TYPE "UDT_WSVStatistics"
VERSION : 0.1
   STRUCT
      "010" { ExternalAccessible := 'False'; ExternalVisible := 'False'; ExternalWritable := 'False'} : Struct
         Conveyor { ExternalAccessible := 'False'; ExternalVisible := 'False'; ExternalWritable := 'False'; S7_SetPoint := 'False'} : "UDT_ConveyorStatistics";
         MCO_M01 { ExternalAccessible := 'False'; ExternalVisible := 'False'; ExternalWritable := 'False'; S7_SetPoint := 'False'} : "UDT_VfdStatistics";
      END_STRUCT;
      "020" { ExternalAccessible := 'False'; ExternalVisible := 'False'; ExternalWritable := 'False'} : Struct
         Conveyor { ExternalAccessible := 'False'; ExternalVisible := 'False'; ExternalWritable := 'False'; S7_SetPoint := 'False'} : "UDT_ConveyorStatistics";
         PEC_Eos { ExternalAccessible := 'False'; ExternalVisible := 'False'; ExternalWritable := 'False'} : "UDT_PECStatistics";
         MCO_M01 { ExternalAccessible := 'False'; ExternalVisible := 'False'; ExternalWritable := 'False'; S7_SetPoint := 'False'} : "UDT_VfdStatistics";
      END_STRUCT;
      "030" { ExternalAccessible := 'False'; ExternalVisible := 'False'; ExternalWritable := 'False'} : Struct
         Conveyor { ExternalAccessible := 'False'; ExternalVisible := 'False'; ExternalWritable := 'False'; S7_SetPoint := 'False'} : "UDT_ConveyorStatistics";
         PEC_Eos { ExternalAccessible := 'False'; ExternalVisible := 'False'; ExternalWritable := 'False'} : "UDT_PECStatistics";
         MCO_M01 { ExternalAccessible := 'False'; ExternalVisible := 'False'; ExternalWritable := 'False'; S7_SetPoint := 'False'} : "UDT_VfdStatistics";
      END_STRUCT;
      "040" { ExternalAccessible := 'False'; ExternalVisible := 'False'; ExternalWritable := 'False'} : Struct
         Conveyor { ExternalAccessible := 'False'; ExternalVisible := 'False'; ExternalWritable := 'False'; S7_SetPoint := 'False'} : "UDT_ConveyorStatistics";
         PEC_Eos { ExternalAccessible := 'False'; ExternalVisible := 'False'; ExternalWritable := 'False'} : "UDT_PECStatistics";
         MCO_M01 { ExternalAccessible := 'False'; ExternalVisible := 'False'; ExternalWritable := 'False'; S7_SetPoint := 'False'} : "UDT_VfdStatistics";
      END_STRUCT;
      "050" { ExternalAccessible := 'False'; ExternalVisible := 'False'; ExternalWritable := 'False'} : Struct
         Conveyor { ExternalAccessible := 'False'; ExternalVisible := 'False'; ExternalWritable := 'False'; S7_SetPoint := 'False'} : "UDT_ConveyorStatistics";
         PEC_Eos { ExternalAccessible := 'False'; ExternalVisible := 'False'; ExternalWritable := 'False'} : "UDT_PECStatistics";
         MCO_M01 { ExternalAccessible := 'False'; ExternalVisible := 'False'; ExternalWritable := 'False'; S7_SetPoint := 'False'} : "UDT_VfdStatistics";
      END_STRUCT;
      "060" { ExternalAccessible := 'False'; ExternalVisible := 'False'; ExternalWritable := 'False'} : Struct
         Conveyor { ExternalAccessible := 'False'; ExternalVisible := 'False'; ExternalWritable := 'False'; S7_SetPoint := 'False'} : "UDT_ConveyorStatistics";
         PEC_Eos { ExternalAccessible := 'False'; ExternalVisible := 'False'; ExternalWritable := 'False'} : "UDT_PECStatistics";
         MCO_M01 { ExternalAccessible := 'False'; ExternalVisible := 'False'; ExternalWritable := 'False'; S7_SetPoint := 'False'} : "UDT_VfdStatistics";
      END_STRUCT;
      "070" { ExternalAccessible := 'False'; ExternalVisible := 'False'; ExternalWritable := 'False'} : Struct
         Conveyor { ExternalAccessible := 'False'; ExternalVisible := 'False'; ExternalWritable := 'False'; S7_SetPoint := 'False'} : "UDT_ConveyorStatistics";
         PEC_Eos { ExternalAccessible := 'False'; ExternalVisible := 'False'; ExternalWritable := 'False'} : "UDT_PECStatistics";
         MCO_M01 { ExternalAccessible := 'False'; ExternalVisible := 'False'; ExternalWritable := 'False'; S7_SetPoint := 'False'} : "UDT_VfdStatistics";
      END_STRUCT;
      "080" { ExternalAccessible := 'False'; ExternalVisible := 'False'; ExternalWritable := 'False'} : Struct
         Conveyor { ExternalAccessible := 'False'; ExternalVisible := 'False'; ExternalWritable := 'False'; S7_SetPoint := 'False'} : "UDT_ConveyorStatistics";
         PEC_Eos { ExternalAccessible := 'False'; ExternalVisible := 'False'; ExternalWritable := 'False'} : "UDT_PECStatistics";
         MCO_M01 { ExternalAccessible := 'False'; ExternalVisible := 'False'; ExternalWritable := 'False'; S7_SetPoint := 'False'} : "UDT_VfdStatistics";
      END_STRUCT;
      "090" { ExternalAccessible := 'False'; ExternalVisible := 'False'; ExternalWritable := 'False'} : Struct
         Conveyor { ExternalAccessible := 'False'; ExternalVisible := 'False'; ExternalWritable := 'False'; S7_SetPoint := 'False'} : "UDT_ConveyorStatistics";
         MCO_M01 { ExternalAccessible := 'False'; ExternalVisible := 'False'; ExternalWritable := 'False'; S7_SetPoint := 'False'} : "UDT_VfdStatistics";
      END_STRUCT;
      "100" { ExternalAccessible := 'False'; ExternalVisible := 'False'; ExternalWritable := 'False'} : Struct
         Conveyor { ExternalAccessible := 'False'; ExternalVisible := 'False'; ExternalWritable := 'False'; S7_SetPoint := 'False'} : "UDT_ConveyorStatistics";
         PEC_Eos { ExternalAccessible := 'False'; ExternalVisible := 'False'; ExternalWritable := 'False'} : "UDT_PECStatistics";
         MCO_M01 { ExternalAccessible := 'False'; ExternalVisible := 'False'; ExternalWritable := 'False'; S7_SetPoint := 'False'} : "UDT_VfdStatistics";
      END_STRUCT;
      "110" { ExternalAccessible := 'False'; ExternalVisible := 'False'; ExternalWritable := 'False'} : Struct
         Conveyor { ExternalAccessible := 'False'; ExternalVisible := 'False'; ExternalWritable := 'False'; S7_SetPoint := 'False'} : "UDT_ConveyorStatistics";
         PEC_Eos { ExternalAccessible := 'False'; ExternalVisible := 'False'; ExternalWritable := 'False'} : "UDT_PECStatistics";
         MCO_M01 { ExternalAccessible := 'False'; ExternalVisible := 'False'; ExternalWritable := 'False'; S7_SetPoint := 'False'} : "UDT_VfdStatistics";
      END_STRUCT;
      "120" { ExternalAccessible := 'False'; ExternalVisible := 'False'; ExternalWritable := 'False'} : Struct
         Conveyor { ExternalAccessible := 'False'; ExternalVisible := 'False'; ExternalWritable := 'False'; S7_SetPoint := 'False'} : "UDT_ConveyorStatistics";
         PEC_Eos { ExternalAccessible := 'False'; ExternalVisible := 'False'; ExternalWritable := 'False'} : "UDT_PECStatistics";
         MCO_M01 { ExternalAccessible := 'False'; ExternalVisible := 'False'; ExternalWritable := 'False'; S7_SetPoint := 'False'} : "UDT_VfdStatistics";
      END_STRUCT;
      "121" { ExternalAccessible := 'False'; ExternalVisible := 'False'; ExternalWritable := 'False'} : Struct
         RightAngledTransfer { ExternalAccessible := 'False'; ExternalVisible := 'False'; ExternalWritable := 'False'; S7_SetPoint := 'False'} : "UDT_RATStatistics";
         MCO_M01 { ExternalAccessible := 'False'; ExternalVisible := 'False'; ExternalWritable := 'False'} : "UDT_VfdStatistics";
      END_STRUCT;
      "230" { ExternalAccessible := 'False'; ExternalVisible := 'False'; ExternalWritable := 'False'} : Struct
         Conveyor { ExternalAccessible := 'False'; ExternalVisible := 'False'; ExternalWritable := 'False'; S7_SetPoint := 'False'} : "UDT_ConveyorStatistics";
         PEC_Eos { ExternalAccessible := 'False'; ExternalVisible := 'False'; ExternalWritable := 'False'} : "UDT_PECUpdateStatistics";
         MCO_M01 { ExternalAccessible := 'False'; ExternalVisible := 'False'; ExternalWritable := 'False'; S7_SetPoint := 'False'} : "UDT_VfdStatistics";
      END_STRUCT;
      "240" { ExternalAccessible := 'False'; ExternalVisible := 'False'; ExternalWritable := 'False'} : Struct
         Conveyor { ExternalAccessible := 'False'; ExternalVisible := 'False'; ExternalWritable := 'False'; S7_SetPoint := 'False'} : "UDT_ConveyorStatistics";
         PEC_Eos { ExternalAccessible := 'False'; ExternalVisible := 'False'; ExternalWritable := 'False'; S7_SetPoint := 'False'} : "UDT_PECStatistics";
         MCO_M01 { ExternalAccessible := 'False'; ExternalVisible := 'False'; ExternalWritable := 'False'; S7_SetPoint := 'False'} : "UDT_VfdStatistics";
      END_STRUCT;
      "241" { ExternalAccessible := 'False'; ExternalVisible := 'False'; ExternalWritable := 'False'} : Struct
         RightAngledTransfer { ExternalAccessible := 'False'; ExternalVisible := 'False'; ExternalWritable := 'False'} : "UDT_RATStatistics";
         MCO_M01 { ExternalAccessible := 'False'; ExternalVisible := 'False'; ExternalWritable := 'False'} : "UDT_VfdStatistics";
      END_STRUCT;
      "250" { ExternalAccessible := 'False'; ExternalVisible := 'False'; ExternalWritable := 'False'} : Struct
         Conveyor { ExternalAccessible := 'False'; ExternalVisible := 'False'; ExternalWritable := 'False'} : "UDT_ConveyorStatistics";
         PEC_EoS { ExternalAccessible := 'False'; ExternalVisible := 'False'; ExternalWritable := 'False'; S7_SetPoint := 'False'} : "UDT_PECUpdateStatistics";
         MCO_M01 { ExternalAccessible := 'False'; ExternalVisible := 'False'; ExternalWritable := 'False'; S7_SetPoint := 'False'} : "UDT_VfdStatistics";
      END_STRUCT;
      "260" { ExternalAccessible := 'False'; ExternalVisible := 'False'; ExternalWritable := 'False'} : Struct
         Conveyor { ExternalAccessible := 'False'; ExternalVisible := 'False'; ExternalWritable := 'False'} : "UDT_ConveyorStatistics";
         VFD { ExternalAccessible := 'False'; ExternalVisible := 'False'; ExternalWritable := 'False'; S7_SetPoint := 'False'} : "UDT_VfdStatistics";
      END_STRUCT;
      "270" { ExternalAccessible := 'False'; ExternalVisible := 'False'; ExternalWritable := 'False'} : Struct
         Conveyor { ExternalAccessible := 'False'; ExternalVisible := 'False'; ExternalWritable := 'False'} : "UDT_ConveyorStatistics";
         PEC_EoS { ExternalAccessible := 'False'; ExternalVisible := 'False'; ExternalWritable := 'False'; S7_SetPoint := 'False'} : "UDT_PECStatistics";
         MCO_M01 { ExternalAccessible := 'False'; ExternalVisible := 'False'; ExternalWritable := 'False'; S7_SetPoint := 'False'} : "UDT_VfdStatistics";
      END_STRUCT;
      "280" { ExternalAccessible := 'False'; ExternalVisible := 'False'; ExternalWritable := 'False'} : Struct
         Conveyor { ExternalAccessible := 'False'; ExternalVisible := 'False'; ExternalWritable := 'False'} : "UDT_ConveyorStatistics";
         PEC_EoS { ExternalAccessible := 'False'; ExternalVisible := 'False'; ExternalWritable := 'False'; S7_SetPoint := 'False'} : "UDT_PECStatistics";
         MCO_M01 { ExternalAccessible := 'False'; ExternalVisible := 'False'; ExternalWritable := 'False'} : "UDT_VfdStatistics";
      END_STRUCT;
      "310" { ExternalAccessible := 'False'; ExternalVisible := 'False'; ExternalWritable := 'False'} : Struct
         Conveyor { ExternalAccessible := 'False'; ExternalVisible := 'False'; ExternalWritable := 'False'; S7_SetPoint := 'False'} : "UDT_ConveyorStatistics";
         VFD { ExternalAccessible := 'False'; ExternalVisible := 'False'; ExternalWritable := 'False'; S7_SetPoint := 'False'} : "UDT_VfdStatistics";
      END_STRUCT;
      "320" { ExternalAccessible := 'False'; ExternalVisible := 'False'; ExternalWritable := 'False'} : Struct
         Conveyor { ExternalAccessible := 'False'; ExternalVisible := 'False'; ExternalWritable := 'False'; S7_SetPoint := 'False'} : "UDT_ConveyorStatistics";
         PEC_Eos { ExternalAccessible := 'False'; ExternalVisible := 'False'; ExternalWritable := 'False'} : "UDT_PECUpdateStatistics";
         MCO_M01 { ExternalAccessible := 'False'; ExternalVisible := 'False'; ExternalWritable := 'False'; S7_SetPoint := 'False'} : "UDT_VfdStatistics";
      END_STRUCT;
      "330" { ExternalAccessible := 'False'; ExternalVisible := 'False'; ExternalWritable := 'False'} : Struct
         Conveyor { ExternalAccessible := 'False'; ExternalVisible := 'False'; ExternalWritable := 'False'; S7_SetPoint := 'False'} : "UDT_ConveyorStatistics";
         PEC_Eos { ExternalAccessible := 'False'; ExternalVisible := 'False'; ExternalWritable := 'False'} : "UDT_PECUpdateStatistics";
         MCO_M01 { ExternalAccessible := 'False'; ExternalVisible := 'False'; ExternalWritable := 'False'} : "UDT_VfdStatistics";
      END_STRUCT;
      "340" { ExternalAccessible := 'False'; ExternalVisible := 'False'; ExternalWritable := 'False'} : Struct
         Conveyor { ExternalAccessible := 'False'; ExternalVisible := 'False'; ExternalWritable := 'False'; S7_SetPoint := 'False'} : "UDT_ConveyorStatistics";
         PEC_Eos { ExternalAccessible := 'False'; ExternalVisible := 'False'; ExternalWritable := 'False'} : "UDT_PECStatistics";
         MCO_M01 { ExternalAccessible := 'False'; ExternalVisible := 'False'; ExternalWritable := 'False'; S7_SetPoint := 'False'} : "UDT_VfdStatistics";
      END_STRUCT;
      "341" { ExternalAccessible := 'False'; ExternalVisible := 'False'; ExternalWritable := 'False'} : Struct
         RightAngledTransfer { ExternalAccessible := 'False'; ExternalVisible := 'False'; ExternalWritable := 'False'; S7_SetPoint := 'False'} : "UDT_RATStatistics";
         MCO_M01 { ExternalAccessible := 'False'; ExternalVisible := 'False'; ExternalWritable := 'False'} : "UDT_VfdStatistics";
      END_STRUCT;
      "350" { ExternalAccessible := 'False'; ExternalVisible := 'False'; ExternalWritable := 'False'} : Struct
         Conveyor { ExternalAccessible := 'False'; ExternalVisible := 'False'; ExternalWritable := 'False'; S7_SetPoint := 'False'} : "UDT_ConveyorStatistics";
         PEC_Eos { ExternalAccessible := 'False'; ExternalVisible := 'False'; ExternalWritable := 'False'} : "UDT_PECStatistics";
         MCO_M01 { ExternalAccessible := 'False'; ExternalVisible := 'False'; ExternalWritable := 'False'; S7_SetPoint := 'False'} : "UDT_VfdStatistics";
      END_STRUCT;
      "351" { ExternalAccessible := 'False'; ExternalVisible := 'False'; ExternalWritable := 'False'} : Struct
         RightAngledTransfer { ExternalAccessible := 'False'; ExternalVisible := 'False'; ExternalWritable := 'False'; S7_SetPoint := 'False'} : "UDT_RATStatistics";
         MCO_M01 { ExternalAccessible := 'False'; ExternalVisible := 'False'; ExternalWritable := 'False'} : "UDT_VfdStatistics";
      END_STRUCT;
      "360" { ExternalAccessible := 'False'; ExternalVisible := 'False'; ExternalWritable := 'False'} : Struct
         Conveyor { ExternalAccessible := 'False'; ExternalVisible := 'False'; ExternalWritable := 'False'; S7_SetPoint := 'False'} : "UDT_ConveyorStatistics";
         PEC_Eos { ExternalAccessible := 'False'; ExternalVisible := 'False'; ExternalWritable := 'False'} : "UDT_PECStatistics";
         MCO_M01 { ExternalAccessible := 'False'; ExternalVisible := 'False'; ExternalWritable := 'False'; S7_SetPoint := 'False'} : "UDT_VfdStatistics";
      END_STRUCT;
      "361" { ExternalAccessible := 'False'; ExternalVisible := 'False'; ExternalWritable := 'False'} : Struct
         RightAngledTransfer { ExternalAccessible := 'False'; ExternalVisible := 'False'; ExternalWritable := 'False'; S7_SetPoint := 'False'} : "UDT_RATStatistics";
         MCO_M01 { ExternalAccessible := 'False'; ExternalVisible := 'False'; ExternalWritable := 'False'} : "UDT_VfdStatistics";
      END_STRUCT;
      "370" { ExternalAccessible := 'False'; ExternalVisible := 'False'; ExternalWritable := 'False'} : Struct
         Conveyor { ExternalAccessible := 'False'; ExternalVisible := 'False'; ExternalWritable := 'False'; S7_SetPoint := 'False'} : "UDT_ConveyorStatistics";
         PEC_Eos { ExternalAccessible := 'False'; ExternalVisible := 'False'; ExternalWritable := 'False'} : "UDT_PECStatistics";
         MCO_M01 { ExternalAccessible := 'False'; ExternalVisible := 'False'; ExternalWritable := 'False'; S7_SetPoint := 'False'} : "UDT_VfdStatistics";
      END_STRUCT;
      "371" { ExternalAccessible := 'False'; ExternalVisible := 'False'; ExternalWritable := 'False'} : Struct
         RightAngledTransfer { ExternalAccessible := 'False'; ExternalVisible := 'False'; ExternalWritable := 'False'; S7_SetPoint := 'False'} : "UDT_RATStatistics";
         MCO_M01 { ExternalAccessible := 'False'; ExternalVisible := 'False'; ExternalWritable := 'False'} : "UDT_VfdStatistics";
      END_STRUCT;
      "380" { ExternalAccessible := 'False'; ExternalVisible := 'False'; ExternalWritable := 'False'} : Struct
         Conveyor { ExternalAccessible := 'False'; ExternalVisible := 'False'; ExternalWritable := 'False'; S7_SetPoint := 'False'} : "UDT_ConveyorStatistics";
         PEC_Eos { ExternalAccessible := 'False'; ExternalVisible := 'False'; ExternalWritable := 'False'} : "UDT_PECUpdateStatistics";
         MCO_M01 { ExternalAccessible := 'False'; ExternalVisible := 'False'; ExternalWritable := 'False'; S7_SetPoint := 'False'} : "UDT_VfdStatistics";
      END_STRUCT;
      "390" { ExternalAccessible := 'False'; ExternalVisible := 'False'; ExternalWritable := 'False'} : Struct
         Conveyor { ExternalAccessible := 'False'; ExternalVisible := 'False'; ExternalWritable := 'False'; S7_SetPoint := 'False'} : "UDT_ConveyorStatistics";
         PEC_Eos { ExternalAccessible := 'False'; ExternalVisible := 'False'; ExternalWritable := 'False'} : "UDT_PECUpdateStatistics";
         MCO_M01 { ExternalAccessible := 'False'; ExternalVisible := 'False'; ExternalWritable := 'False'; S7_SetPoint := 'False'} : "UDT_VfdStatistics";
      END_STRUCT;
      "530" { ExternalAccessible := 'False'; ExternalVisible := 'False'; ExternalWritable := 'False'} : Struct
         Conveyor { ExternalAccessible := 'False'; ExternalVisible := 'False'; ExternalWritable := 'False'; S7_SetPoint := 'False'} : "UDT_ConveyorStatistics";
         PEC_Eos { ExternalAccessible := 'False'; ExternalVisible := 'False'; ExternalWritable := 'False'} : "UDT_PECUpdateStatistics";
         MCO_M01 { ExternalAccessible := 'False'; ExternalVisible := 'False'; ExternalWritable := 'False'; S7_SetPoint := 'False'} : "UDT_VfdStatistics";
      END_STRUCT;
      "540" { ExternalAccessible := 'False'; ExternalVisible := 'False'; ExternalWritable := 'False'} : Struct
         Conveyor { ExternalAccessible := 'False'; ExternalVisible := 'False'; ExternalWritable := 'False'; S7_SetPoint := 'False'} : "UDT_ConveyorStatistics";
         PEC_Eos { ExternalAccessible := 'False'; ExternalVisible := 'False'; ExternalWritable := 'False'; S7_SetPoint := 'False'} : "UDT_PECStatistics";
         MCO_M01 { ExternalAccessible := 'False'; ExternalVisible := 'False'; ExternalWritable := 'False'; S7_SetPoint := 'False'} : "UDT_VfdStatistics";
      END_STRUCT;
      "541" { ExternalAccessible := 'False'; ExternalVisible := 'False'; ExternalWritable := 'False'} : Struct
         RightAngledTransfer { ExternalAccessible := 'False'; ExternalVisible := 'False'; ExternalWritable := 'False'} : "UDT_RATStatistics";
         MCO_M01 { ExternalAccessible := 'False'; ExternalVisible := 'False'; ExternalWritable := 'False'} : "UDT_VfdStatistics";
      END_STRUCT;
      "550" { ExternalAccessible := 'False'; ExternalVisible := 'False'; ExternalWritable := 'False'} : Struct
         Conveyor { ExternalAccessible := 'False'; ExternalVisible := 'False'; ExternalWritable := 'False'} : "UDT_ConveyorStatistics";
         PEC_EoS { ExternalAccessible := 'False'; ExternalVisible := 'False'; ExternalWritable := 'False'; S7_SetPoint := 'False'} : "UDT_PECUpdateStatistics";
         MCO_M01 { ExternalAccessible := 'False'; ExternalVisible := 'False'; ExternalWritable := 'False'; S7_SetPoint := 'False'} : "UDT_VfdStatistics";
      END_STRUCT;
      "560" { ExternalAccessible := 'False'; ExternalVisible := 'False'; ExternalWritable := 'False'} : Struct
         Conveyor { ExternalAccessible := 'False'; ExternalVisible := 'False'; ExternalWritable := 'False'} : "UDT_ConveyorStatistics";
         VFD { ExternalAccessible := 'False'; ExternalVisible := 'False'; ExternalWritable := 'False'; S7_SetPoint := 'False'} : "UDT_VfdStatistics";
      END_STRUCT;
      "570" { ExternalAccessible := 'False'; ExternalVisible := 'False'; ExternalWritable := 'False'} : Struct
         Conveyor { ExternalAccessible := 'False'; ExternalVisible := 'False'; ExternalWritable := 'False'} : "UDT_ConveyorStatistics";
         PEC_EoS { ExternalAccessible := 'False'; ExternalVisible := 'False'; ExternalWritable := 'False'; S7_SetPoint := 'False'} : "UDT_PECStatistics";
         MCO_M01 { ExternalAccessible := 'False'; ExternalVisible := 'False'; ExternalWritable := 'False'; S7_SetPoint := 'False'} : "UDT_VfdStatistics";
      END_STRUCT;
      "580" { ExternalAccessible := 'False'; ExternalVisible := 'False'; ExternalWritable := 'False'} : Struct
         Conveyor { ExternalAccessible := 'False'; ExternalVisible := 'False'; ExternalWritable := 'False'} : "UDT_ConveyorStatistics";
         PEC_EoS { ExternalAccessible := 'False'; ExternalVisible := 'False'; ExternalWritable := 'False'; S7_SetPoint := 'False'} : "UDT_PECStatistics";
         MCO_M01 { ExternalAccessible := 'False'; ExternalVisible := 'False'; ExternalWritable := 'False'} : "UDT_VfdStatistics";
      END_STRUCT;
      "610" { ExternalAccessible := 'False'; ExternalVisible := 'False'; ExternalWritable := 'False'} : Struct
         Conveyor { ExternalAccessible := 'False'; ExternalVisible := 'False'; ExternalWritable := 'False'; S7_SetPoint := 'False'} : "UDT_ConveyorStatistics";
         VFD { ExternalAccessible := 'False'; ExternalVisible := 'False'; ExternalWritable := 'False'; S7_SetPoint := 'False'} : "UDT_VfdStatistics";
      END_STRUCT;
      "620" { ExternalAccessible := 'False'; ExternalVisible := 'False'; ExternalWritable := 'False'} : Struct
         Conveyor { ExternalAccessible := 'False'; ExternalVisible := 'False'; ExternalWritable := 'False'; S7_SetPoint := 'False'} : "UDT_ConveyorStatistics";
         PEC_Eos { ExternalAccessible := 'False'; ExternalVisible := 'False'; ExternalWritable := 'False'} : "UDT_PECUpdateStatistics";
         MCO_M01 { ExternalAccessible := 'False'; ExternalVisible := 'False'; ExternalWritable := 'False'; S7_SetPoint := 'False'} : "UDT_VfdStatistics";
      END_STRUCT;
      "630" { ExternalAccessible := 'False'; ExternalVisible := 'False'; ExternalWritable := 'False'} : Struct
         Conveyor { ExternalAccessible := 'False'; ExternalVisible := 'False'; ExternalWritable := 'False'; S7_SetPoint := 'False'} : "UDT_ConveyorStatistics";
         PEC_Eos { ExternalAccessible := 'False'; ExternalVisible := 'False'; ExternalWritable := 'False'} : "UDT_PECUpdateStatistics";
         MCO_M01 { ExternalAccessible := 'False'; ExternalVisible := 'False'; ExternalWritable := 'False'} : "UDT_VfdStatistics";
      END_STRUCT;
      "640" { ExternalAccessible := 'False'; ExternalVisible := 'False'; ExternalWritable := 'False'} : Struct
         Conveyor { ExternalAccessible := 'False'; ExternalVisible := 'False'; ExternalWritable := 'False'; S7_SetPoint := 'False'} : "UDT_ConveyorStatistics";
         PEC_Eos { ExternalAccessible := 'False'; ExternalVisible := 'False'; ExternalWritable := 'False'} : "UDT_PECStatistics";
         MCO_M01 { ExternalAccessible := 'False'; ExternalVisible := 'False'; ExternalWritable := 'False'; S7_SetPoint := 'False'} : "UDT_VfdStatistics";
      END_STRUCT;
      "641" { ExternalAccessible := 'False'; ExternalVisible := 'False'; ExternalWritable := 'False'} : Struct
         RightAngledTransfer { ExternalAccessible := 'False'; ExternalVisible := 'False'; ExternalWritable := 'False'; S7_SetPoint := 'False'} : "UDT_RATStatistics";
         MCO_M01 { ExternalAccessible := 'False'; ExternalVisible := 'False'; ExternalWritable := 'False'} : "UDT_VfdStatistics";
      END_STRUCT;
      "650" { ExternalAccessible := 'False'; ExternalVisible := 'False'; ExternalWritable := 'False'} : Struct
         Conveyor { ExternalAccessible := 'False'; ExternalVisible := 'False'; ExternalWritable := 'False'; S7_SetPoint := 'False'} : "UDT_ConveyorStatistics";
         PEC_Eos { ExternalAccessible := 'False'; ExternalVisible := 'False'; ExternalWritable := 'False'} : "UDT_PECStatistics";
         MCO_M01 { ExternalAccessible := 'False'; ExternalVisible := 'False'; ExternalWritable := 'False'} : "UDT_VfdStatistics";
      END_STRUCT;
      "651" { ExternalAccessible := 'False'; ExternalVisible := 'False'; ExternalWritable := 'False'} : Struct
         RightAngledTransfer { ExternalAccessible := 'False'; ExternalVisible := 'False'; ExternalWritable := 'False'; S7_SetPoint := 'False'} : "UDT_RATStatistics";
         MCO_M01 { ExternalAccessible := 'False'; ExternalVisible := 'False'; ExternalWritable := 'False'} : "UDT_VfdStatistics";
      END_STRUCT;
      "660" { ExternalAccessible := 'False'; ExternalVisible := 'False'; ExternalWritable := 'False'} : Struct
         Conveyor { ExternalAccessible := 'False'; ExternalVisible := 'False'; ExternalWritable := 'False'; S7_SetPoint := 'False'} : "UDT_ConveyorStatistics";
         PEC_Eos { ExternalAccessible := 'False'; ExternalVisible := 'False'; ExternalWritable := 'False'} : "UDT_PECStatistics";
         MCO_M01 { ExternalAccessible := 'False'; ExternalVisible := 'False'; ExternalWritable := 'False'; S7_SetPoint := 'False'} : "UDT_VfdStatistics";
      END_STRUCT;
      "661" { ExternalAccessible := 'False'; ExternalVisible := 'False'; ExternalWritable := 'False'} : Struct
         RightAngledTransfer { ExternalAccessible := 'False'; ExternalVisible := 'False'; ExternalWritable := 'False'; S7_SetPoint := 'False'} : "UDT_RATStatistics";
         MCO_M01 { ExternalAccessible := 'False'; ExternalVisible := 'False'; ExternalWritable := 'False'} : "UDT_VfdStatistics";
      END_STRUCT;
      "670" { ExternalAccessible := 'False'; ExternalVisible := 'False'; ExternalWritable := 'False'} : Struct
         Conveyor { ExternalAccessible := 'False'; ExternalVisible := 'False'; ExternalWritable := 'False'; S7_SetPoint := 'False'} : "UDT_ConveyorStatistics";
         PEC_Eos { ExternalAccessible := 'False'; ExternalVisible := 'False'; ExternalWritable := 'False'} : "UDT_PECStatistics";
         MCO_M01 { ExternalAccessible := 'False'; ExternalVisible := 'False'; ExternalWritable := 'False'; S7_SetPoint := 'False'} : "UDT_VfdStatistics";
      END_STRUCT;
      "671" { ExternalAccessible := 'False'; ExternalVisible := 'False'; ExternalWritable := 'False'} : Struct
         RightAngledTransfer { ExternalAccessible := 'False'; ExternalVisible := 'False'; ExternalWritable := 'False'; S7_SetPoint := 'False'} : "UDT_RATStatistics";
         MCO_M01 { ExternalAccessible := 'False'; ExternalVisible := 'False'; ExternalWritable := 'False'} : "UDT_VfdStatistics";
      END_STRUCT;
      "680" { ExternalAccessible := 'False'; ExternalVisible := 'False'; ExternalWritable := 'False'} : Struct
         Conveyor { ExternalAccessible := 'False'; ExternalVisible := 'False'; ExternalWritable := 'False'; S7_SetPoint := 'False'} : "UDT_ConveyorStatistics";
         PEC_Eos { ExternalAccessible := 'False'; ExternalVisible := 'False'; ExternalWritable := 'False'} : "UDT_PECUpdateStatistics";
         MCO_M01 { ExternalAccessible := 'False'; ExternalVisible := 'False'; ExternalWritable := 'False'; S7_SetPoint := 'False'} : "UDT_VfdStatistics";
      END_STRUCT;
      "690" { ExternalAccessible := 'False'; ExternalVisible := 'False'; ExternalWritable := 'False'} : Struct
         Conveyor { ExternalAccessible := 'False'; ExternalVisible := 'False'; ExternalWritable := 'False'; S7_SetPoint := 'False'} : "UDT_ConveyorStatistics";
         PEC_Eos { ExternalAccessible := 'False'; ExternalVisible := 'False'; ExternalWritable := 'False'} : "UDT_PECUpdateStatistics";
         MCO_M01 { ExternalAccessible := 'False'; ExternalVisible := 'False'; ExternalWritable := 'False'; S7_SetPoint := 'False'} : "UDT_VfdStatistics";
      END_STRUCT;
   END_STRUCT;

END_TYPE

FUNCTION_BLOCK "FB_Valve"
TITLE = Single ended Valve Control and monitor
{ S7_Optimized_Access := 'TRUE' }
AUTHOR : 'I.Ajram'
VERSION : 0.1
   VAR_INPUT
      iUDT_Configuration { ExternalAccessible := 'False'; ExternalVisible := 'False'; ExternalWritable := 'False'} : "UDT_ValveConfiguration";   // Valve configuration
      ix_Open { ExternalAccessible := 'False'; ExternalVisible := 'False'; ExternalWritable := 'False'} : Bool;   // Open command (Hold if ControlMode = 1, pulse if ControlMode = 2)
      ix_Close { ExternalAccessible := 'False'; ExternalVisible := 'False'; ExternalWritable := 'False'} : Bool;   // Close command (Not used if ControlMode = 1, pulse if ControlMode = 2)
      ix_IsOpened { ExternalAccessible := 'False'; ExternalVisible := 'False'; ExternalWritable := 'False'} : Bool;   // Feedback Signal ( Not used if #iqUDT_SEVConfiguration.IsOpenFeedBackExist is FALSE)
      ix_IsClosed { ExternalAccessible := 'False'; ExternalVisible := 'False'; ExternalWritable := 'False'} : Bool;   // Feedback Signal ( Not used if #iqUDT_SEVConfiguration.IsCloseFeedBackExist is FALSE)
      ix_AirPressureOk { ExternalAccessible := 'False'; ExternalVisible := 'False'; ExternalWritable := 'False'} : Bool;   // Air pressure is healthy
   END_VAR

   VAR_OUTPUT
      qx_Open { ExternalAccessible := 'False'; ExternalVisible := 'False'; ExternalWritable := 'False'} : Bool;   // Open command
      qx_Close { ExternalAccessible := 'False'; ExternalVisible := 'False'; ExternalWritable := 'False'} : Bool;   // Close command
      qUDT_HMIStatus { ExternalAccessible := 'False'; ExternalVisible := 'False'; ExternalWritable := 'False'} : "UDT_ValveStatus";
      qUDT_Statistics { ExternalAccessible := 'False'; ExternalVisible := 'False'; ExternalWritable := 'False'} : "UDT_ValveStatistics";
   END_VAR

   VAR_IN_OUT
      iqUDT_HMICommand : "UDT_ValveCommand";   // Interafce for HMI commands
      iqUDT_Interface : "UDT_ValveInterface";   // Interface with external modules
      iqUDT_EquipmentControl : "UDT_EquipmentControl";   // Equipment control structure
   END_VAR

   VAR
      sx_ManualModeSelected { ExternalAccessible := 'False'; ExternalVisible := 'False'; ExternalWritable := 'False'} : Bool;
      sx_AutoModeSelected { ExternalAccessible := 'False'; ExternalVisible := 'False'; ExternalWritable := 'False'} : Bool;
      sx_OpenActivated { ExternalAccessible := 'False'; ExternalVisible := 'False'; ExternalWritable := 'False'} : Bool;
      sx_CloseActivated { ExternalAccessible := 'False'; ExternalVisible := 'False'; ExternalWritable := 'False'} : Bool;
      sx_FaultActive { ExternalAccessible := 'False'; ExternalVisible := 'False'; ExternalWritable := 'False'} : Bool;
      sTON_Opening {InstructionName := 'TON_TIME'; LibVersion := '1.0'; ExternalAccessible := 'False'; ExternalVisible := 'False'; ExternalWritable := 'False'; S7_SetPoint := 'False'} : TON_TIME;
      sTON_Closing {InstructionName := 'TON_TIME'; LibVersion := '1.0'; ExternalAccessible := 'False'; ExternalVisible := 'False'; ExternalWritable := 'False'; S7_SetPoint := 'False'} : TON_TIME;
      sTime_Closing { ExternalAccessible := 'False'; ExternalVisible := 'False'; ExternalWritable := 'False'} : Time;
      sTime_Opening { ExternalAccessible := 'False'; ExternalVisible := 'False'; ExternalWritable := 'False'} : Time;
      RTRIG_Open {InstructionName := 'R_TRIG'; LibVersion := '1.0'; ExternalAccessible := 'False'; ExternalVisible := 'False'; ExternalWritable := 'False'; S7_SetPoint := 'False'} : R_TRIG;
      RTRIG_Close {InstructionName := 'R_TRIG'; LibVersion := '1.0'; ExternalAccessible := 'False'; ExternalVisible := 'False'; ExternalWritable := 'False'; S7_SetPoint := 'False'} : R_TRIG;
      RTRIG_FaultActive {InstructionName := 'R_TRIG'; LibVersion := '1.0'; ExternalAccessible := 'False'; ExternalVisible := 'False'; ExternalWritable := 'False'; S7_SetPoint := 'False'} : R_TRIG;
      RTRIG_Opened {InstructionName := 'R_TRIG'; LibVersion := '1.0'; ExternalAccessible := 'False'; ExternalVisible := 'False'; ExternalWritable := 'False'; S7_SetPoint := 'False'} : R_TRIG;
   END_VAR

   VAR CONSTANT
      ci_ControlModeHold : Int := 1;   // Energize to hold
      ci_ControlModePulse : Int := 2;   // Pulse energized to change state
      ci_ValveTypeSEV : Int := 1;   // Single coil valve
      ci_ValveTypeDEV : Int := 2;   // Double coil valve, bi-stable, latching
   END_VAR


BEGIN
	(*
	----------------------------------------------------------------------------------------

	Version history:
	Date        | Version   | Author        | Remark
	----------------------------------------------------------------------------------------
	08/07/2024  | 0.1       | I. Ajram      | first release TIA 18
	16/07/2024  | 0.2       | I. Ajram      | Changed block name from FB_SEV to FB_Valve
	                                        |  +    Added Configuration to allow for SEV and DEV
	                                        |  +    Added qx_Close Output
	                                        |  +    Added logic to accomodate for DEV
	30/08/2024  | 0.3       | J. Majer      | Added comments, number regions, added iq_UDT_EquipmentInterface, iqUDT_EquipmentControl
	----------------------------------------------------------------------------------------

	*)

	REGION 1 - Edge detection
	    // Trigger rising edge detection for different signals: Open, Close, FaultActive, and Opened.
	    #RTRIG_Open(CLK := #ix_Open OR #iqUDT_Interface.Open);
	    #RTRIG_Close(CLK := #ix_Close OR #iqUDT_Interface.Close);
	    #RTRIG_FaultActive(CLK := #sx_FaultActive);
	    #RTRIG_Opened(CLK := #qUDT_HMIStatus.Specific.Opened);

	END_REGION

	REGION 2 - Auto / Manual

	    // Handle auto mode command.
	    IF #iqUDT_EquipmentControl.Command.Start AND #iqUDT_EquipmentControl.Command.AutomaticOn
	    THEN
	        #sx_AutoModeSelected := TRUE;
	        #sx_ManualModeSelected := FALSE;
	        #iqUDT_HMICommand.AutoMode := FALSE;
	    END_IF;

	    // Manual mode bits inputs can be reset in case of malfunction
	    IF #iqUDT_EquipmentControl.Command.DisableManualMode
	    THEN
	        #iqUDT_HMICommand.ManualMode := FALSE;
	        #iqUDT_EquipmentControl.Command.ManualMode := FALSE;
	    END_IF;

	    // Handle manual mode command.
	    IF (#iqUDT_EquipmentControl.Command.ManualMode OR #iqUDT_HMICommand.ManualMode)
	        AND NOT #iqUDT_EquipmentControl.Command.DisableManualMode
	    THEN
	        #sx_AutoModeSelected := FALSE;
	        #sx_ManualModeSelected := TRUE;
	        #iqUDT_HMICommand.ManualMode := FALSE;
	    END_IF;

	    REGION 2.1 - Restart request

	        // Indicating need for system restart if no mode is selected
	        #iqUDT_EquipmentControl.Request.RestartRequired := NOT #sx_AutoModeSelected
	        AND NOT #sx_AutoModeSelected;

	    END_REGION
	END_REGION

	REGION 3 - Faults

	    REGION 3.1 - Configuration Error
	        // Check for configuration errors by validating the ControlMode and ValveType values.
	        IF #iUDT_Configuration.ControlMode < #ci_ControlModeHold
	            OR #iUDT_Configuration.ControlMode > #ci_ControlModePulse
	            OR #iUDT_Configuration.ValveType < #ci_ValveTypeSEV
	            OR #iUDT_Configuration.ValveType > #ci_ValveTypeDEV
	        THEN
	            #qUDT_HMIStatus.Specific.ConfigurationError := TRUE;
	        ELSE
	            #qUDT_HMIStatus.Specific.ConfigurationError := FALSE;
	        END_IF;

	    END_REGION

	    REGION 3.2 - Low Pressure
	        // Set AirPressureLost flag if air pressure is not okay.
	        IF NOT #ix_AirPressureOk THEN
	            #qUDT_HMIStatus.Specific.AirPressureLost := TRUE;
	        END_IF;

	    END_REGION

	    REGION 3.3 - Fail to Open
	        // Set FailToOpen flag if the valve failed to open within the expected time.
	        IF #sTON_Opening.Q AND #iUDT_Configuration.OpenFeedBackExist THEN
	            #qUDT_HMIStatus.Specific.FailToOpen := TRUE;
	        END_IF;

	    END_REGION

	    REGION 3.4 - Fail to Close
	        // Set FailToClose flag if the valve failed to close within the expected time.
	        IF #sTON_Closing.Q AND #iUDT_Configuration.CloseFeedBackExist THEN
	            #qUDT_HMIStatus.Specific.FailToClose := TRUE;
	        END_IF;

	    END_REGION

	    REGION 3.4 - Collective fault
	        // Set FaultActive flag if any specific fault is detected (fail to open/close, air pressure lost, or configuration error).
	        #sx_FaultActive := #qUDT_HMIStatus.Specific.FailToClose OR
	        #qUDT_HMIStatus.Specific.FailToOpen OR
	        #qUDT_HMIStatus.Specific.AirPressureLost OR
	        #qUDT_HMIStatus.Specific.ConfigurationError;

	        // forward error to the interface with other modules
	        #iqUDT_Interface.Error := #sx_FaultActive;

	        // If FaultActive is set, deactivate open and close commands.
	        IF #sx_FaultActive THEN
	            #sx_OpenActivated := FALSE;
	            #sx_CloseActivated := FALSE;
	        END_IF;

	    END_REGION

	    REGION 3.5 - Reset
	        // Reset fault flags and set air pressure flag based on the state of AirPressureOk.
	        IF #iqUDT_EquipmentControl.Command.Reset THEN
	            #qUDT_HMIStatus.Specific.FailToOpen := FALSE;
	            #qUDT_HMIStatus.Specific.FailToClose := FALSE;
	            #qUDT_HMIStatus.Specific.AirPressureLost := NOT #ix_AirPressureOk;
	        END_IF;

	    END_REGION

	END_REGION

	REGION 4 - Command
	    // Process commands based on the current mode (Auto/Manual) and fault state.
	    IF NOT #sx_FaultActive THEN

	        REGION 4.1 - Auto
	            // Handle command logic in Auto mode based on control mode (Hold or Pulse).
	            IF #sx_AutoModeSelected THEN
	                CASE #iUDT_Configuration.ControlMode OF

	                        // ControlModeHold: Open/close based on the ix_Open signal.
	                    #ci_ControlModeHold:
	                        #sx_OpenActivated := #ix_Open;
	                        #sx_CloseActivated := NOT #ix_Open;

	                        // ControlModePulse: Open/close based on rising edge detection.
	                    #ci_ControlModePulse:
	                        IF #RTRIG_Open.Q AND NOT #ix_IsOpened THEN
	                            #sx_OpenActivated := TRUE;
	                            #sx_CloseActivated := FALSE;
	                        END_IF;

	                        IF #RTRIG_Close.Q AND NOT #ix_IsClosed THEN
	                            #sx_OpenActivated := FALSE;
	                            #sx_CloseActivated := TRUE;
	                        END_IF;

	                END_CASE;
	            END_IF;

	        END_REGION

	        REGION 4.2 - Manual
	            // Handle command logic in Manual mode based on control mode (Hold or Pulse).
	            IF #sx_ManualModeSelected THEN
	                CASE #iUDT_Configuration.ControlMode OF

	                        // ControlModeHold: Open/close based on manual commands.
	                    #ci_ControlModeHold:
	                        #sx_OpenActivated := #iqUDT_HMICommand.ManualOpen;
	                        #sx_CloseActivated := #iqUDT_HMICommand.ManualClose;

	                        // ControlModePulse: Open/close based on manual commands with feedback checks.
	                    #ci_ControlModePulse:
	                        IF #iqUDT_HMICommand.ManualOpen AND NOT #ix_IsOpened THEN
	                            #sx_OpenActivated := TRUE;
	                            #sx_CloseActivated := FALSE;
	                            #iqUDT_HMICommand.ManualOpen := FALSE;
	                        END_IF;

	                        IF #iqUDT_HMICommand.ManualClose AND NOT #ix_IsClosed THEN
	                            #sx_OpenActivated := FALSE;
	                            #sx_CloseActivated := TRUE;
	                            #iqUDT_HMICommand.ManualClose := FALSE;
	                        END_IF;

	                END_CASE;
	            END_IF;

	        END_REGION
	    ELSE
	        // On fault, clear all open/close commands.
	        #sx_OpenActivated := FALSE;
	        #sx_CloseActivated := FALSE;
	        #iqUDT_HMICommand.ManualClose := FALSE;
	        #iqUDT_HMICommand.ManualOpen := FALSE;
	    END_IF;

	END_REGION

	REGION 5 - Statistics
	    // Update statistical data when reset or fault occurs.
	    IF #iqUDT_EquipmentControl.Command.ResetData OR #sx_FaultActive THEN
	        "FC_Statistics"(ix_Reset := #iqUDT_EquipmentControl.Command.ResetData,
	                        ix_Activate := #sx_FaultActive,
	                        ix_RTrigActivate := #RTRIG_FaultActive.Q,
	                        iqUDT_Statistics := #qUDT_Statistics.Fail);
	    END_IF;

	    // Update open statistics when reset or opened.
	    IF #iqUDT_EquipmentControl.Command.ResetData OR #qUDT_HMIStatus.Specific.Opened THEN
	        "FC_Statistics"(ix_Reset := #iqUDT_EquipmentControl.Command.ResetData,
	                        ix_Activate := #qUDT_HMIStatus.Specific.Opened,
	                        ix_RTrigActivate := #RTRIG_Opened.Q,
	                        iqUDT_Statistics := #qUDT_Statistics.Open);
	    END_IF;

	END_REGION

	REGION 6 - Status

	    REGION 6.1 - Opened / Closed
	        // Handle open/close status based on feedback or timers.
	        IF #iUDT_Configuration.OpenFeedBackExist THEN
	            // Set opened status based on feedback.
	            #qUDT_HMIStatus.Specific.Opened := #ix_IsOpened;
	        ELSE
	            // Use opening timer as an indicator if feedback is not available.
	            IF #sTON_Opening.Q THEN
	                #qUDT_HMIStatus.Specific.Opened := TRUE;
	            END_IF;
	            IF #sx_CloseActivated THEN
	                #qUDT_HMIStatus.Specific.Opened := FALSE;
	            END_IF;
	        END_IF;

	        // Module interface valve feedback opened
	        #iqUDT_Interface.IsOpened := #qUDT_HMIStatus.Specific.Opened;

	        IF #iUDT_Configuration.CloseFeedBackExist THEN
	            // Set closed status based on feedback.
	            #qUDT_HMIStatus.Specific.Closed := #ix_IsClosed;
	        ELSE
	            // Use closing timer as an indicator if feedback is not available.
	            IF #sTON_Closing.Q THEN
	                #qUDT_HMIStatus.Specific.Closed := TRUE;
	            END_IF;
	            IF #sx_OpenActivated THEN
	                #qUDT_HMIStatus.Specific.Closed := FALSE;
	            END_IF;
	        END_IF;

	        // Module interface valve feedback closed
	        #iqUDT_Interface.IsClosed := #qUDT_HMIStatus.Specific.Closed;

	    END_REGION

	    REGION 6.2 - Opening
	        // Handle the logic for the valve opening, including timer initialization and status updates.
	        IF #iUDT_Configuration.OpenTime = 0 THEN
	            #sTime_Opening := T#1s;  // Default to 1 second if not configured.
	        ELSE
	            #sTime_Opening := INT_TO_TIME(#iUDT_Configuration.OpenTime);  // Use configured open time.
	        END_IF;

	        IF #sx_OpenActivated AND NOT #qUDT_HMIStatus.Specific.Opened THEN
	            #qUDT_HMIStatus.Specific.Opening := TRUE;
	        ELSE
	            #qUDT_HMIStatus.Specific.Opening := FALSE;
	        END_IF;

	        // Start the opening timer.
	        #sTON_Opening(IN := #qUDT_HMIStatus.Specific.Opening,
	                      PT := #sTime_Opening);

	    END_REGION

	    REGION 6.3 - Closing
	        // Handle the logic for the valve closing, including timer initialization and status updates.
	        IF #iUDT_Configuration.CloseTime = 0 THEN
	            #sTime_Closing := T#1s;  // Default to 1 second if not configured.
	        ELSE
	            #sTime_Closing := INT_TO_TIME(#iUDT_Configuration.CloseTime);  // Use configured close time.
	        END_IF;

	        IF #sx_CloseActivated AND NOT #qUDT_HMIStatus.Specific.Closed THEN
	            #qUDT_HMIStatus.Specific.Closing := TRUE;
	        ELSE
	            #qUDT_HMIStatus.Specific.Closing := FALSE;
	        END_IF;

	        // Start the closing timer.
	        #sTON_Closing(IN := #qUDT_HMIStatus.Specific.Closing,
	                      PT := #sTime_Closing);

	    END_REGION

	END_REGION

	REGION 7 - Output

	    // Select the action based on the valve type configuration
	    CASE #iUDT_Configuration.ValveType OF

	            // SEV Valve Type
	        #ci_ValveTypeSEV:
	            // The valve opens if Open is activated, Close is not activated, and no fault is active
	            #qx_Open :=
	            #sx_OpenActivated AND
	            NOT #sx_CloseActivated AND
	            NOT #sx_FaultActive;

	            // Reset the open signal, SEV logic requires manual reset after operation
	            #qx_Open := FALSE;

	            // DEV Valve Type
	        #ci_ValveTypeDEV:
	            // The valve opens if there are no faults, Open is activated, and the valve is not yet opened
	            #qx_Open :=
	            NOT #sx_FaultActive AND
	            #sx_OpenActivated AND NOT #qUDT_HMIStatus.Specific.Opened;

	            // The valve closes if there are no faults, Close is activated, and the valve is not yet closed
	            #qx_Close :=
	            NOT #sx_FaultActive AND
	            #sx_CloseActivated AND NOT #qUDT_HMIStatus.Specific.Closed;

	            // If the valve is opened, a fault occurs, or the valve is in the closing state, deactivate Open
	            IF #qUDT_HMIStatus.Specific.Opened OR
	                #sx_FaultActive OR
	                #qUDT_HMIStatus.Specific.Closing
	            THEN
	                #sx_OpenActivated := FALSE;
	            END_IF;

	            // If the valve is closed, a fault occurs, or the valve is in the opening state, deactivate Close
	            IF #qUDT_HMIStatus.Specific.Closed OR
	                #sx_FaultActive OR
	                #qUDT_HMIStatus.Specific.Opening
	            THEN
	                #sx_CloseActivated := FALSE;
	            END_IF;

	    END_CASE;

	END_REGION

END_FUNCTION_BLOCK

TYPE "UDT_TGWLiftCommonStatus"
VERSION : 0.1
   STRUCT
      "010" { S7_SetPoint := 'False'} : "UDT_CommonStatus";
      "020" { S7_SetPoint := 'False'} : "UDT_CommonStatus";
   END_STRUCT;

END_TYPE

TYPE "UDT_WSVStatus"
VERSION : 0.1
   STRUCT
      "010" { ExternalAccessible := 'False'; ExternalVisible := 'False'; ExternalWritable := 'False'} : Struct
         Conveyor { ExternalAccessible := 'False'; ExternalVisible := 'False'; ExternalWritable := 'False'; S7_SetPoint := 'False'} : "UDT_ConveyorStatus";
         MCO_M01 { ExternalAccessible := 'False'; ExternalVisible := 'False'; ExternalWritable := 'False'} : "UDT_AixControllerStatus";
      END_STRUCT;
      "020" { ExternalAccessible := 'False'; ExternalVisible := 'False'; ExternalWritable := 'False'} : Struct
         Conveyor { ExternalAccessible := 'False'; ExternalVisible := 'False'; ExternalWritable := 'False'; S7_SetPoint := 'False'} : "UDT_ConveyorStatus";
         PEC_Eos { ExternalAccessible := 'False'; ExternalVisible := 'False'; ExternalWritable := 'False'} : "UDT_PECStatus";
         MCO_M01 { ExternalAccessible := 'False'; ExternalVisible := 'False'; ExternalWritable := 'False'} : "UDT_AixControllerStatus";
      END_STRUCT;
      "030" { ExternalAccessible := 'False'; ExternalVisible := 'False'; ExternalWritable := 'False'} : Struct
         Conveyor { ExternalAccessible := 'False'; ExternalVisible := 'False'; ExternalWritable := 'False'; S7_SetPoint := 'False'} : "UDT_ConveyorStatus";
         PEC_Eos { ExternalAccessible := 'False'; ExternalVisible := 'False'; ExternalWritable := 'False'} : "UDT_PECStatus";
         MCO_M01 { ExternalAccessible := 'False'; ExternalVisible := 'False'; ExternalWritable := 'False'} : "UDT_AixControllerStatus";
      END_STRUCT;
      "040" { ExternalAccessible := 'False'; ExternalVisible := 'False'; ExternalWritable := 'False'} : Struct
         Conveyor { ExternalAccessible := 'False'; ExternalVisible := 'False'; ExternalWritable := 'False'; S7_SetPoint := 'False'} : "UDT_ConveyorStatus";
         PEC_Eos { ExternalAccessible := 'False'; ExternalVisible := 'False'; ExternalWritable := 'False'} : "UDT_PECStatus";
         MCO_M01 { ExternalAccessible := 'False'; ExternalVisible := 'False'; ExternalWritable := 'False'} : "UDT_AixControllerStatus";
      END_STRUCT;
      "050" { ExternalAccessible := 'False'; ExternalVisible := 'False'; ExternalWritable := 'False'} : Struct
         Conveyor { ExternalAccessible := 'False'; ExternalVisible := 'False'; ExternalWritable := 'False'; S7_SetPoint := 'False'} : "UDT_ConveyorStatus";
         PEC_Eos { ExternalAccessible := 'False'; ExternalVisible := 'False'; ExternalWritable := 'False'} : "UDT_PECStatus";
         MCO_M01 { ExternalAccessible := 'False'; ExternalVisible := 'False'; ExternalWritable := 'False'} : "UDT_AixControllerStatus";
      END_STRUCT;
      "060" { ExternalAccessible := 'False'; ExternalVisible := 'False'; ExternalWritable := 'False'} : Struct
         Conveyor { ExternalAccessible := 'False'; ExternalVisible := 'False'; ExternalWritable := 'False'; S7_SetPoint := 'False'} : "UDT_ConveyorStatus";
         PEC_Eos { ExternalAccessible := 'False'; ExternalVisible := 'False'; ExternalWritable := 'False'} : "UDT_PECStatus";
         MCO_M01 { ExternalAccessible := 'False'; ExternalVisible := 'False'; ExternalWritable := 'False'} : "UDT_AixControllerStatus";
      END_STRUCT;
      "070" { ExternalAccessible := 'False'; ExternalVisible := 'False'; ExternalWritable := 'False'} : Struct
         Conveyor { ExternalAccessible := 'False'; ExternalVisible := 'False'; ExternalWritable := 'False'; S7_SetPoint := 'False'} : "UDT_ConveyorStatus";
         PEC_Eos { ExternalAccessible := 'False'; ExternalVisible := 'False'; ExternalWritable := 'False'} : "UDT_PECStatus";
         MCO_M01 { ExternalAccessible := 'False'; ExternalVisible := 'False'; ExternalWritable := 'False'} : "UDT_AixControllerStatus";
      END_STRUCT;
      "080" { ExternalAccessible := 'False'; ExternalVisible := 'False'; ExternalWritable := 'False'} : Struct
         Conveyor { ExternalAccessible := 'False'; ExternalVisible := 'False'; ExternalWritable := 'False'; S7_SetPoint := 'False'} : "UDT_ConveyorStatus";
         PEC_Eos { ExternalAccessible := 'False'; ExternalVisible := 'False'; ExternalWritable := 'False'} : "UDT_PECStatus";
         MCO_M01 { ExternalAccessible := 'False'; ExternalVisible := 'False'; ExternalWritable := 'False'} : "UDT_AixControllerStatus";
      END_STRUCT;
      "090" { ExternalAccessible := 'False'; ExternalVisible := 'False'; ExternalWritable := 'False'} : Struct
         Conveyor { ExternalAccessible := 'False'; ExternalVisible := 'False'; ExternalWritable := 'False'; S7_SetPoint := 'False'} : "UDT_ConveyorStatus";
         MCO_M01 { ExternalAccessible := 'False'; ExternalVisible := 'False'; ExternalWritable := 'False'} : "UDT_AixControllerStatus";
      END_STRUCT;
      "100" { ExternalAccessible := 'False'; ExternalVisible := 'False'; ExternalWritable := 'False'} : Struct
         Conveyor { ExternalAccessible := 'False'; ExternalVisible := 'False'; ExternalWritable := 'False'; S7_SetPoint := 'False'} : "UDT_ConveyorStatus";
         PEC_Eos { ExternalAccessible := 'False'; ExternalVisible := 'False'; ExternalWritable := 'False'} : "UDT_PECStatus";
         MCO_M01 { ExternalAccessible := 'False'; ExternalVisible := 'False'; ExternalWritable := 'False'} : "UDT_AixControllerStatus";
      END_STRUCT;
      "110" { ExternalAccessible := 'False'; ExternalVisible := 'False'; ExternalWritable := 'False'} : Struct
         Conveyor { ExternalAccessible := 'False'; ExternalVisible := 'False'; ExternalWritable := 'False'; S7_SetPoint := 'False'} : "UDT_ConveyorStatus";
         PEC_Eos { ExternalAccessible := 'False'; ExternalVisible := 'False'; ExternalWritable := 'False'} : "UDT_PECStatus";
         MCO_M01 { ExternalAccessible := 'False'; ExternalVisible := 'False'; ExternalWritable := 'False'} : "UDT_AixControllerStatus";
      END_STRUCT;
      "120" { ExternalAccessible := 'False'; ExternalVisible := 'False'; ExternalWritable := 'False'} : Struct
         Conveyor { ExternalAccessible := 'False'; ExternalVisible := 'False'; ExternalWritable := 'False'; S7_SetPoint := 'False'} : "UDT_ConveyorStatus";
         PEC_Eos { ExternalAccessible := 'False'; ExternalVisible := 'False'; ExternalWritable := 'False'} : "UDT_PECStatus";
         MCO_M01 { ExternalAccessible := 'False'; ExternalVisible := 'False'; ExternalWritable := 'False'} : "UDT_AixControllerStatus";
      END_STRUCT;
      "121" { ExternalAccessible := 'False'; ExternalVisible := 'False'; ExternalWritable := 'False'} : Struct
         RightAngledTransfer { ExternalAccessible := 'False'; ExternalVisible := 'False'; ExternalWritable := 'False'; S7_SetPoint := 'False'} : "UDT_RATStatus";
         MCO_M01 { ExternalAccessible := 'False'; ExternalVisible := 'False'; ExternalWritable := 'False'} : "UDT_AixControllerStatus";
      END_STRUCT;
      "230" { ExternalAccessible := 'False'; ExternalVisible := 'False'; ExternalWritable := 'False'} : Struct
         Conveyor { ExternalAccessible := 'False'; ExternalVisible := 'False'; ExternalWritable := 'False'; S7_SetPoint := 'False'} : "UDT_ConveyorStatus";
         PEC_Eos { ExternalAccessible := 'False'; ExternalVisible := 'False'; ExternalWritable := 'False'} : "UDT_PECUpdateStatus";
         MCO_M01 { ExternalAccessible := 'False'; ExternalVisible := 'False'; ExternalWritable := 'False'} : "UDT_AixControllerStatus";
      END_STRUCT;
      "240" { ExternalAccessible := 'False'; ExternalVisible := 'False'; ExternalWritable := 'False'} : Struct
         Conveyor { ExternalAccessible := 'False'; ExternalVisible := 'False'; ExternalWritable := 'False'; S7_SetPoint := 'False'} : "UDT_ConveyorStatus";
         PEC_Eos { ExternalAccessible := 'False'; ExternalVisible := 'False'; ExternalWritable := 'False'; S7_SetPoint := 'False'} : "UDT_PECStatus";
         MCO_M01 { ExternalAccessible := 'False'; ExternalVisible := 'False'; ExternalWritable := 'False'; S7_SetPoint := 'False'} : "UDT_AixControllerStatus";
      END_STRUCT;
      "241" { ExternalAccessible := 'False'; ExternalVisible := 'False'; ExternalWritable := 'False'} : Struct
         RightAngledTransfer { ExternalAccessible := 'False'; ExternalVisible := 'False'; ExternalWritable := 'False'} : "UDT_RATStatus";
         MCO_M01 { ExternalAccessible := 'False'; ExternalVisible := 'False'; ExternalWritable := 'False'} : "UDT_AixControllerStatus";
      END_STRUCT;
      "250" { ExternalAccessible := 'False'; ExternalVisible := 'False'; ExternalWritable := 'False'} : Struct
         Conveyor { ExternalAccessible := 'False'; ExternalVisible := 'False'; ExternalWritable := 'False'} : "UDT_ConveyorStatus";
         PEC_EoS { ExternalAccessible := 'False'; ExternalVisible := 'False'; ExternalWritable := 'False'; S7_SetPoint := 'False'} : "UDT_PECUpdateStatus";
         MCO_M01 { ExternalAccessible := 'False'; ExternalVisible := 'False'; ExternalWritable := 'False'} : "UDT_AixControllerStatus";
      END_STRUCT;
      "260" { ExternalAccessible := 'False'; ExternalVisible := 'False'; ExternalWritable := 'False'} : Struct
         Conveyor { ExternalAccessible := 'False'; ExternalVisible := 'False'; ExternalWritable := 'False'} : "UDT_ConveyorStatus";
         VFD { ExternalAccessible := 'False'; ExternalVisible := 'False'; ExternalWritable := 'False'} : "UDT_VfdStatus";
      END_STRUCT;
      "270" { ExternalAccessible := 'False'; ExternalVisible := 'False'; ExternalWritable := 'False'} : Struct
         Conveyor { ExternalAccessible := 'False'; ExternalVisible := 'False'; ExternalWritable := 'False'} : "UDT_ConveyorStatus";
         PEC_EoS { ExternalAccessible := 'False'; ExternalVisible := 'False'; ExternalWritable := 'False'; S7_SetPoint := 'False'} : "UDT_PECStatus";
         MCO_M01 { ExternalAccessible := 'False'; ExternalVisible := 'False'; ExternalWritable := 'False'} : "UDT_AixControllerStatus";
      END_STRUCT;
      "280" { ExternalAccessible := 'False'; ExternalVisible := 'False'; ExternalWritable := 'False'} : Struct
         Conveyor { ExternalAccessible := 'False'; ExternalVisible := 'False'; ExternalWritable := 'False'} : "UDT_ConveyorStatus";
         PEC_EoS { ExternalAccessible := 'False'; ExternalVisible := 'False'; ExternalWritable := 'False'; S7_SetPoint := 'False'} : "UDT_PECStatus";
         MCO_M01 { ExternalAccessible := 'False'; ExternalVisible := 'False'; ExternalWritable := 'False'} : "UDT_AixControllerStatus";
      END_STRUCT;
      "310" { ExternalAccessible := 'False'; ExternalVisible := 'False'; ExternalWritable := 'False'} : Struct
         Conveyor { ExternalAccessible := 'False'; ExternalVisible := 'False'; ExternalWritable := 'False'; S7_SetPoint := 'False'} : "UDT_ConveyorStatus";
         VFD { ExternalAccessible := 'False'; ExternalVisible := 'False'; ExternalWritable := 'False'} : "UDT_VfdStatus";
      END_STRUCT;
      "320" { ExternalAccessible := 'False'; ExternalVisible := 'False'; ExternalWritable := 'False'} : Struct
         Conveyor { ExternalAccessible := 'False'; ExternalVisible := 'False'; ExternalWritable := 'False'; S7_SetPoint := 'False'} : "UDT_ConveyorStatus";
         PEC_Eos { ExternalAccessible := 'False'; ExternalVisible := 'False'; ExternalWritable := 'False'} : "UDT_PECUpdateStatus";
         MCO_M01 { ExternalAccessible := 'False'; ExternalVisible := 'False'; ExternalWritable := 'False'} : "UDT_AixControllerStatus";
      END_STRUCT;
      "330" { ExternalAccessible := 'False'; ExternalVisible := 'False'; ExternalWritable := 'False'} : Struct
         Conveyor { ExternalAccessible := 'False'; ExternalVisible := 'False'; ExternalWritable := 'False'; S7_SetPoint := 'False'} : "UDT_ConveyorStatus";
         PEC_Eos { ExternalAccessible := 'False'; ExternalVisible := 'False'; ExternalWritable := 'False'} : "UDT_PECUpdateStatus";
         MCO_M01 { ExternalAccessible := 'False'; ExternalVisible := 'False'; ExternalWritable := 'False'} : "UDT_AixControllerStatus";
      END_STRUCT;
      "340" { ExternalAccessible := 'False'; ExternalVisible := 'False'; ExternalWritable := 'False'} : Struct
         Conveyor { ExternalAccessible := 'False'; ExternalVisible := 'False'; ExternalWritable := 'False'; S7_SetPoint := 'False'} : "UDT_ConveyorStatus";
         PEC_Eos { ExternalAccessible := 'False'; ExternalVisible := 'False'; ExternalWritable := 'False'} : "UDT_PECStatus";
         MCO_M01 { ExternalAccessible := 'False'; ExternalVisible := 'False'; ExternalWritable := 'False'} : "UDT_AixControllerStatus";
      END_STRUCT;
      "341" { ExternalAccessible := 'False'; ExternalVisible := 'False'; ExternalWritable := 'False'} : Struct
         RightAngledTransfer { ExternalAccessible := 'False'; ExternalVisible := 'False'; ExternalWritable := 'False'; S7_SetPoint := 'False'} : "UDT_RATStatus";
         MCO_M01 { ExternalAccessible := 'False'; ExternalVisible := 'False'; ExternalWritable := 'False'} : "UDT_AixControllerStatus";
      END_STRUCT;
      "350" { ExternalAccessible := 'False'; ExternalVisible := 'False'; ExternalWritable := 'False'} : Struct
         Conveyor { ExternalAccessible := 'False'; ExternalVisible := 'False'; ExternalWritable := 'False'; S7_SetPoint := 'False'} : "UDT_ConveyorStatus";
         PEC_Eos { ExternalAccessible := 'False'; ExternalVisible := 'False'; ExternalWritable := 'False'} : "UDT_PECStatus";
         MCO_M01 { ExternalAccessible := 'False'; ExternalVisible := 'False'; ExternalWritable := 'False'} : "UDT_AixControllerStatus";
      END_STRUCT;
      "351" { ExternalAccessible := 'False'; ExternalVisible := 'False'; ExternalWritable := 'False'} : Struct
         RightAngledTransfer { ExternalAccessible := 'False'; ExternalVisible := 'False'; ExternalWritable := 'False'; S7_SetPoint := 'False'} : "UDT_RATStatus";
         MCO_M01 { ExternalAccessible := 'False'; ExternalVisible := 'False'; ExternalWritable := 'False'} : "UDT_AixControllerStatus";
      END_STRUCT;
      "360" { ExternalAccessible := 'False'; ExternalVisible := 'False'; ExternalWritable := 'False'} : Struct
         Conveyor { ExternalAccessible := 'False'; ExternalVisible := 'False'; ExternalWritable := 'False'; S7_SetPoint := 'False'} : "UDT_ConveyorStatus";
         PEC_Eos { ExternalAccessible := 'False'; ExternalVisible := 'False'; ExternalWritable := 'False'} : "UDT_PECStatus";
         MCO_M01 { ExternalAccessible := 'False'; ExternalVisible := 'False'; ExternalWritable := 'False'} : "UDT_AixControllerStatus";
      END_STRUCT;
      "361" { ExternalAccessible := 'False'; ExternalVisible := 'False'; ExternalWritable := 'False'} : Struct
         RightAngledTransfer { ExternalAccessible := 'False'; ExternalVisible := 'False'; ExternalWritable := 'False'; S7_SetPoint := 'False'} : "UDT_RATStatus";
         MCO_M01 { ExternalAccessible := 'False'; ExternalVisible := 'False'; ExternalWritable := 'False'} : "UDT_AixControllerStatus";
      END_STRUCT;
      "370" { ExternalAccessible := 'False'; ExternalVisible := 'False'; ExternalWritable := 'False'} : Struct
         Conveyor { ExternalAccessible := 'False'; ExternalVisible := 'False'; ExternalWritable := 'False'; S7_SetPoint := 'False'} : "UDT_ConveyorStatus";
         PEC_Eos { ExternalAccessible := 'False'; ExternalVisible := 'False'; ExternalWritable := 'False'} : "UDT_PECStatus";
         MCO_M01 { ExternalAccessible := 'False'; ExternalVisible := 'False'; ExternalWritable := 'False'} : "UDT_AixControllerStatus";
      END_STRUCT;
      "371" { ExternalAccessible := 'False'; ExternalVisible := 'False'; ExternalWritable := 'False'} : Struct
         RightAngledTransfer { ExternalAccessible := 'False'; ExternalVisible := 'False'; ExternalWritable := 'False'; S7_SetPoint := 'False'} : "UDT_RATStatus";
         MCO_M01 { ExternalAccessible := 'False'; ExternalVisible := 'False'; ExternalWritable := 'False'} : "UDT_AixControllerStatus";
      END_STRUCT;
      "380" { ExternalAccessible := 'False'; ExternalVisible := 'False'; ExternalWritable := 'False'} : Struct
         Conveyor { ExternalAccessible := 'False'; ExternalVisible := 'False'; ExternalWritable := 'False'; S7_SetPoint := 'False'} : "UDT_ConveyorStatus";
         PEC_Eos { ExternalAccessible := 'False'; ExternalVisible := 'False'; ExternalWritable := 'False'} : "UDT_PECUpdateStatus";
         MCO_M01 { ExternalAccessible := 'False'; ExternalVisible := 'False'; ExternalWritable := 'False'} : "UDT_AixControllerStatus";
      END_STRUCT;
      "390" { ExternalAccessible := 'False'; ExternalVisible := 'False'; ExternalWritable := 'False'} : Struct
         Conveyor { ExternalAccessible := 'False'; ExternalVisible := 'False'; ExternalWritable := 'False'; S7_SetPoint := 'False'} : "UDT_ConveyorStatus";
         PEC_Eos { ExternalAccessible := 'False'; ExternalVisible := 'False'; ExternalWritable := 'False'} : "UDT_PECUpdateStatus";
         MCO_M01 { ExternalAccessible := 'False'; ExternalVisible := 'False'; ExternalWritable := 'False'} : "UDT_AixControllerStatus";
      END_STRUCT;
      "530" { ExternalAccessible := 'False'; ExternalVisible := 'False'; ExternalWritable := 'False'} : Struct
         Conveyor { ExternalAccessible := 'False'; ExternalVisible := 'False'; ExternalWritable := 'False'; S7_SetPoint := 'False'} : "UDT_ConveyorStatus";
         PEC_Eos { ExternalAccessible := 'False'; ExternalVisible := 'False'; ExternalWritable := 'False'} : "UDT_PECUpdateStatus";
         MCO_M01 { ExternalAccessible := 'False'; ExternalVisible := 'False'; ExternalWritable := 'False'} : "UDT_AixControllerStatus";
      END_STRUCT;
      "540" { ExternalAccessible := 'False'; ExternalVisible := 'False'; ExternalWritable := 'False'} : Struct
         Conveyor { ExternalAccessible := 'False'; ExternalVisible := 'False'; ExternalWritable := 'False'; S7_SetPoint := 'False'} : "UDT_ConveyorStatus";
         PEC_Eos { ExternalAccessible := 'False'; ExternalVisible := 'False'; ExternalWritable := 'False'; S7_SetPoint := 'False'} : "UDT_PECStatus";
         MCO_M01 { ExternalAccessible := 'False'; ExternalVisible := 'False'; ExternalWritable := 'False'; S7_SetPoint := 'False'} : "UDT_AixControllerStatus";
      END_STRUCT;
      "541" { ExternalAccessible := 'False'; ExternalVisible := 'False'; ExternalWritable := 'False'} : Struct
         RightAngledTransfer { ExternalAccessible := 'False'; ExternalVisible := 'False'; ExternalWritable := 'False'} : "UDT_RATStatus";
         MCO_M01 { ExternalAccessible := 'False'; ExternalVisible := 'False'; ExternalWritable := 'False'} : "UDT_AixControllerStatus";
      END_STRUCT;
      "550" { ExternalAccessible := 'False'; ExternalVisible := 'False'; ExternalWritable := 'False'} : Struct
         Conveyor { ExternalAccessible := 'False'; ExternalVisible := 'False'; ExternalWritable := 'False'} : "UDT_ConveyorStatus";
         PEC_EoS { ExternalAccessible := 'False'; ExternalVisible := 'False'; ExternalWritable := 'False'; S7_SetPoint := 'False'} : "UDT_PECUpdateStatus";
         MCO_M01 { ExternalAccessible := 'False'; ExternalVisible := 'False'; ExternalWritable := 'False'} : "UDT_AixControllerStatus";
      END_STRUCT;
      "560" { ExternalAccessible := 'False'; ExternalVisible := 'False'; ExternalWritable := 'False'} : Struct
         Conveyor { ExternalAccessible := 'False'; ExternalVisible := 'False'; ExternalWritable := 'False'} : "UDT_ConveyorStatus";
         VFD { ExternalAccessible := 'False'; ExternalVisible := 'False'; ExternalWritable := 'False'} : "UDT_VfdStatus";
      END_STRUCT;
      "570" { ExternalAccessible := 'False'; ExternalVisible := 'False'; ExternalWritable := 'False'} : Struct
         Conveyor { ExternalAccessible := 'False'; ExternalVisible := 'False'; ExternalWritable := 'False'} : "UDT_ConveyorStatus";
         PEC_EoS { ExternalAccessible := 'False'; ExternalVisible := 'False'; ExternalWritable := 'False'; S7_SetPoint := 'False'} : "UDT_PECStatus";
         MCO_M01 { ExternalAccessible := 'False'; ExternalVisible := 'False'; ExternalWritable := 'False'} : "UDT_AixControllerStatus";
      END_STRUCT;
      "580" { ExternalAccessible := 'False'; ExternalVisible := 'False'; ExternalWritable := 'False'} : Struct
         Conveyor { ExternalAccessible := 'False'; ExternalVisible := 'False'; ExternalWritable := 'False'} : "UDT_ConveyorStatus";
         PEC_EoS { ExternalAccessible := 'False'; ExternalVisible := 'False'; ExternalWritable := 'False'; S7_SetPoint := 'False'} : "UDT_PECStatus";
         MCO_M01 { ExternalAccessible := 'False'; ExternalVisible := 'False'; ExternalWritable := 'False'} : "UDT_AixControllerStatus";
      END_STRUCT;
      "610" { ExternalAccessible := 'False'; ExternalVisible := 'False'; ExternalWritable := 'False'} : Struct
         Conveyor { ExternalAccessible := 'False'; ExternalVisible := 'False'; ExternalWritable := 'False'; S7_SetPoint := 'False'} : "UDT_ConveyorStatus";
         VFD { ExternalAccessible := 'False'; ExternalVisible := 'False'; ExternalWritable := 'False'} : "UDT_VfdStatus";
      END_STRUCT;
      "620" { ExternalAccessible := 'False'; ExternalVisible := 'False'; ExternalWritable := 'False'} : Struct
         Conveyor { ExternalAccessible := 'False'; ExternalVisible := 'False'; ExternalWritable := 'False'; S7_SetPoint := 'False'} : "UDT_ConveyorStatus";
         PEC_Eos { ExternalAccessible := 'False'; ExternalVisible := 'False'; ExternalWritable := 'False'} : "UDT_PECUpdateStatus";
         MCO_M01 { ExternalAccessible := 'False'; ExternalVisible := 'False'; ExternalWritable := 'False'} : "UDT_AixControllerStatus";
      END_STRUCT;
      "630" { ExternalAccessible := 'False'; ExternalVisible := 'False'; ExternalWritable := 'False'} : Struct
         Conveyor { ExternalAccessible := 'False'; ExternalVisible := 'False'; ExternalWritable := 'False'; S7_SetPoint := 'False'} : "UDT_ConveyorStatus";
         PEC_Eos { ExternalAccessible := 'False'; ExternalVisible := 'False'; ExternalWritable := 'False'} : "UDT_PECUpdateStatus";
         MCO_M01 { ExternalAccessible := 'False'; ExternalVisible := 'False'; ExternalWritable := 'False'} : "UDT_AixControllerStatus";
      END_STRUCT;
      "640" { ExternalAccessible := 'False'; ExternalVisible := 'False'; ExternalWritable := 'False'} : Struct
         Conveyor { ExternalAccessible := 'False'; ExternalVisible := 'False'; ExternalWritable := 'False'; S7_SetPoint := 'False'} : "UDT_ConveyorStatus";
         PEC_Eos { ExternalAccessible := 'False'; ExternalVisible := 'False'; ExternalWritable := 'False'} : "UDT_PECStatus";
         MCO_M01 { ExternalAccessible := 'False'; ExternalVisible := 'False'; ExternalWritable := 'False'} : "UDT_AixControllerStatus";
      END_STRUCT;
      "641" { ExternalAccessible := 'False'; ExternalVisible := 'False'; ExternalWritable := 'False'} : Struct
         RightAngledTransfer { ExternalAccessible := 'False'; ExternalVisible := 'False'; ExternalWritable := 'False'; S7_SetPoint := 'False'} : "UDT_RATStatus";
         MCO_M01 { ExternalAccessible := 'False'; ExternalVisible := 'False'; ExternalWritable := 'False'} : "UDT_AixControllerStatus";
      END_STRUCT;
      "650" { ExternalAccessible := 'False'; ExternalVisible := 'False'; ExternalWritable := 'False'} : Struct
         Conveyor { ExternalAccessible := 'False'; ExternalVisible := 'False'; ExternalWritable := 'False'; S7_SetPoint := 'False'} : "UDT_ConveyorStatus";
         PEC_Eos { ExternalAccessible := 'False'; ExternalVisible := 'False'; ExternalWritable := 'False'} : "UDT_PECStatus";
         MCO_M01 { ExternalAccessible := 'False'; ExternalVisible := 'False'; ExternalWritable := 'False'} : "UDT_AixControllerStatus";
      END_STRUCT;
      "651" { ExternalAccessible := 'False'; ExternalVisible := 'False'; ExternalWritable := 'False'} : Struct
         RightAngledTransfer { ExternalAccessible := 'False'; ExternalVisible := 'False'; ExternalWritable := 'False'; S7_SetPoint := 'False'} : "UDT_RATStatus";
         MCO_M01 { ExternalAccessible := 'False'; ExternalVisible := 'False'; ExternalWritable := 'False'} : "UDT_AixControllerStatus";
      END_STRUCT;
      "660" { ExternalAccessible := 'False'; ExternalVisible := 'False'; ExternalWritable := 'False'} : Struct
         Conveyor { ExternalAccessible := 'False'; ExternalVisible := 'False'; ExternalWritable := 'False'; S7_SetPoint := 'False'} : "UDT_ConveyorStatus";
         PEC_Eos { ExternalAccessible := 'False'; ExternalVisible := 'False'; ExternalWritable := 'False'} : "UDT_PECStatus";
         MCO_M01 { ExternalAccessible := 'False'; ExternalVisible := 'False'; ExternalWritable := 'False'} : "UDT_AixControllerStatus";
      END_STRUCT;
      "661" { ExternalAccessible := 'False'; ExternalVisible := 'False'; ExternalWritable := 'False'} : Struct
         RightAngledTransfer { ExternalAccessible := 'False'; ExternalVisible := 'False'; ExternalWritable := 'False'; S7_SetPoint := 'False'} : "UDT_RATStatus";
         MCO_M01 { ExternalAccessible := 'False'; ExternalVisible := 'False'; ExternalWritable := 'False'} : "UDT_AixControllerStatus";
      END_STRUCT;
      "670" { ExternalAccessible := 'False'; ExternalVisible := 'False'; ExternalWritable := 'False'} : Struct
         Conveyor { ExternalAccessible := 'False'; ExternalVisible := 'False'; ExternalWritable := 'False'; S7_SetPoint := 'False'} : "UDT_ConveyorStatus";
         PEC_Eos { ExternalAccessible := 'False'; ExternalVisible := 'False'; ExternalWritable := 'False'} : "UDT_PECStatus";
         MCO_M01 { ExternalAccessible := 'False'; ExternalVisible := 'False'; ExternalWritable := 'False'} : "UDT_AixControllerStatus";
      END_STRUCT;
      "671" { ExternalAccessible := 'False'; ExternalVisible := 'False'; ExternalWritable := 'False'} : Struct
         RightAngledTransfer { ExternalAccessible := 'False'; ExternalVisible := 'False'; ExternalWritable := 'False'; S7_SetPoint := 'False'} : "UDT_RATStatus";
         MCO_M01 { ExternalAccessible := 'False'; ExternalVisible := 'False'; ExternalWritable := 'False'} : "UDT_AixControllerStatus";
      END_STRUCT;
      "680" { ExternalAccessible := 'False'; ExternalVisible := 'False'; ExternalWritable := 'False'} : Struct
         Conveyor { ExternalAccessible := 'False'; ExternalVisible := 'False'; ExternalWritable := 'False'; S7_SetPoint := 'False'} : "UDT_ConveyorStatus";
         PEC_Eos { ExternalAccessible := 'False'; ExternalVisible := 'False'; ExternalWritable := 'False'} : "UDT_PECUpdateStatus";
         MCO_M01 { ExternalAccessible := 'False'; ExternalVisible := 'False'; ExternalWritable := 'False'} : "UDT_AixControllerStatus";
      END_STRUCT;
      "690" { ExternalAccessible := 'False'; ExternalVisible := 'False'; ExternalWritable := 'False'} : Struct
         Conveyor { ExternalAccessible := 'False'; ExternalVisible := 'False'; ExternalWritable := 'False'; S7_SetPoint := 'False'} : "UDT_ConveyorStatus";
         PEC_Eos { ExternalAccessible := 'False'; ExternalVisible := 'False'; ExternalWritable := 'False'} : "UDT_PECUpdateStatus";
         MCO_M01 { ExternalAccessible := 'False'; ExternalVisible := 'False'; ExternalWritable := 'False'} : "UDT_AixControllerStatus";
      END_STRUCT;
   END_STRUCT;

END_TYPE

TYPE "UDT_WSVCommonStatus"
VERSION : 0.1
   STRUCT
      "010" { S7_SetPoint := 'False'} : "UDT_CommonStatus";
      "020" { S7_SetPoint := 'False'} : "UDT_CommonStatus";
      "030" { S7_SetPoint := 'False'} : "UDT_CommonStatus";
      "040" { S7_SetPoint := 'False'} : "UDT_CommonStatus";
      "050" { S7_SetPoint := 'False'} : "UDT_CommonStatus";
      "060" { S7_SetPoint := 'False'} : "UDT_CommonStatus";
      "070" { S7_SetPoint := 'False'} : "UDT_CommonStatus";
      "080" { S7_SetPoint := 'False'} : "UDT_CommonStatus";
      "090" { S7_SetPoint := 'False'} : "UDT_CommonStatus";
      "100" { S7_SetPoint := 'False'} : "UDT_CommonStatus";
      "110" { S7_SetPoint := 'False'} : "UDT_CommonStatus";
      "120" { S7_SetPoint := 'False'} : "UDT_CommonStatus";
      "121" { S7_SetPoint := 'False'} : "UDT_CommonStatus";
      "230" { S7_SetPoint := 'False'} : "UDT_CommonStatus";
      "240" { S7_SetPoint := 'False'} : "UDT_CommonStatus";
      "241" { S7_SetPoint := 'False'} : "UDT_CommonStatus";
      "250" { S7_SetPoint := 'False'} : "UDT_CommonStatus";
      "260" { S7_SetPoint := 'False'} : "UDT_CommonStatus";
      "270" { S7_SetPoint := 'False'} : "UDT_CommonStatus";
      "280" { S7_SetPoint := 'False'} : "UDT_CommonStatus";
      "310" { S7_SetPoint := 'False'} : "UDT_CommonStatus";
      "320" { S7_SetPoint := 'False'} : "UDT_CommonStatus";
      "330" { S7_SetPoint := 'False'} : "UDT_CommonStatus";
      "340" { S7_SetPoint := 'False'} : "UDT_CommonStatus";
      "341" { S7_SetPoint := 'False'} : "UDT_CommonStatus";
      "350" { S7_SetPoint := 'False'} : "UDT_CommonStatus";
      "351" { S7_SetPoint := 'False'} : "UDT_CommonStatus";
      "360" { S7_SetPoint := 'False'} : "UDT_CommonStatus";
      "361" { S7_SetPoint := 'False'} : "UDT_CommonStatus";
      "370" { S7_SetPoint := 'False'} : "UDT_CommonStatus";
      "371" { S7_SetPoint := 'False'} : "UDT_CommonStatus";
      "380" { S7_SetPoint := 'False'} : "UDT_CommonStatus";
      "390" { S7_SetPoint := 'False'} : "UDT_CommonStatus";
      "530" { S7_SetPoint := 'False'} : "UDT_CommonStatus";
      "540" { S7_SetPoint := 'False'} : "UDT_CommonStatus";
      "541" { S7_SetPoint := 'False'} : "UDT_CommonStatus";
      "550" { S7_SetPoint := 'False'} : "UDT_CommonStatus";
      "560" { S7_SetPoint := 'False'} : "UDT_CommonStatus";
      "570" { S7_SetPoint := 'False'} : "UDT_CommonStatus";
      "580" { S7_SetPoint := 'False'} : "UDT_CommonStatus";
      "610" { S7_SetPoint := 'False'} : "UDT_CommonStatus";
      "620" { S7_SetPoint := 'False'} : "UDT_CommonStatus";
      "630" { S7_SetPoint := 'False'} : "UDT_CommonStatus";
      "640" { S7_SetPoint := 'False'} : "UDT_CommonStatus";
      "641" { S7_SetPoint := 'False'} : "UDT_CommonStatus";
      "650" { S7_SetPoint := 'False'} : "UDT_CommonStatus";
      "651" { S7_SetPoint := 'False'} : "UDT_CommonStatus";
      "660" { S7_SetPoint := 'False'} : "UDT_CommonStatus";
      "661" { S7_SetPoint := 'False'} : "UDT_CommonStatus";
      "670" { S7_SetPoint := 'False'} : "UDT_CommonStatus";
      "671" { S7_SetPoint := 'False'} : "UDT_CommonStatus";
      "680" { S7_SetPoint := 'False'} : "UDT_CommonStatus";
      "690" { S7_SetPoint := 'False'} : "UDT_CommonStatus";
   END_STRUCT;

END_TYPE

FUNCTION_BLOCK "FB_HMDecode"
TITLE = FB_H&MDecode
{ S7_Optimized_Access := 'TRUE' }
AUTHOR : Fortna
VERSION : 3.0
// ATTRIBUTES
// AUTO_NUMBER = True
// BLOCK_NUMBER = 197
// END_ATTRIBUTES
//Function block to decode H&M messages.
   VAR_INPUT
      II_PLCID { ExternalAccessible := 'False'; ExternalVisible := 'False'; ExternalWritable := 'False'} : Int;   // PLC ID number
   END_VAR

   VAR_OUTPUT
      qx_Error { ExternalAccessible := 'False'; ExternalVisible := 'False'; ExternalWritable := 'False'} : Bool;   // Collective error output
      qx_Warning { ExternalAccessible := 'False'; ExternalVisible := 'False'; ExternalWritable := 'False'} : Bool;   // Collective warning output
   END_VAR

   VAR_IN_OUT
      iqUDT_FifoRcvHeader : "UDT_FifoHeader";   // FIFO receive header
      iqa_FifoRcvData : Array[*] of "UDT_Message";   // FIFO receive data
      iqx_HeartBeat { ExternalAccessible := 'False'; ExternalVisible := 'False'; ExternalWritable := 'False'} : Bool;   // Heartbeat message detect
   END_VAR

   VAR
      sUDT_MessageHeader { ExternalAccessible := 'False'; ExternalVisible := 'False'; ExternalWritable := 'False'; S7_SetPoint := 'False'} : "UDT_HMMessageHeader";
      sUDT_FifoMsg { ExternalAccessible := 'False'; ExternalVisible := 'False'; ExternalWritable := 'False'; S7_SetPoint := 'False'} : "UDT_Message";   // Buffer for fifos message
      sa_Status { ExternalAccessible := 'False'; ExternalVisible := 'False'; ExternalWritable := 'False'} : Struct   // Status structure
         BadMessage { ExternalAccessible := 'False'; ExternalVisible := 'False'; ExternalWritable := 'False'} : Array[1..10] of "UDT_Message";   //   Unknown message read
         FIFORcvStatus { ExternalAccessible := 'False'; ExternalVisible := 'False'; ExternalWritable := 'False'} : "UDT_FifoStatus";   //   Receive FIFO status structure
         FIFOError { ExternalAccessible := 'False'; ExternalVisible := 'False'; ExternalWritable := 'False'; S7_SetPoint := 'True'} : Bool;   //   FIFO error
         FIFOWarning { ExternalAccessible := 'False'; ExternalVisible := 'False'; ExternalWritable := 'False'; S7_SetPoint := 'True'} : Bool;   //   FIFO warning
         AcknowledgeError { ExternalAccessible := 'False'; ExternalVisible := 'False'; ExternalWritable := 'False'; S7_SetPoint := 'True'} : Bool;   //   Acknowledge error
         AcknowledgeWarning { ExternalAccessible := 'False'; ExternalVisible := 'False'; ExternalWritable := 'False'; S7_SetPoint := 'True'} : Bool;   //   Acknowledge warning
         HB_NotOK { ExternalAccessible := 'False'; ExternalVisible := 'False'; ExternalWritable := 'False'} : Bool;   //   Health bit not OK
      END_STRUCT;
      sa_HBRec { ExternalAccessible := 'False'; ExternalVisible := 'False'; ExternalWritable := 'False'} : Struct   // HB message last received timestamp (as string)
         "Date" { ExternalAccessible := 'False'; ExternalVisible := 'False'; ExternalWritable := 'False'} : String;
         "Time" { ExternalAccessible := 'False'; ExternalVisible := 'False'; ExternalWritable := 'False'} : String;
      END_STRUCT;
      sa_DestRec { ExternalAccessible := 'False'; ExternalVisible := 'False'; ExternalWritable := 'False'} : Struct   // Destination message last received timestamp (as string)
         Gin { ExternalAccessible := 'False'; ExternalVisible := 'False'; ExternalWritable := 'False'} : String[4];   // Gin of this product
         Dest1 { ExternalAccessible := 'False'; ExternalVisible := 'False'; ExternalWritable := 'False'} : String[4];   // First possible destination
         Dest2 { ExternalAccessible := 'False'; ExternalVisible := 'False'; ExternalWritable := 'False'} : String[4];   // Second possible destination
         Dest3 { ExternalAccessible := 'False'; ExternalVisible := 'False'; ExternalWritable := 'False'} : String[4];   // Third possible destination
         Dest4 { ExternalAccessible := 'False'; ExternalVisible := 'False'; ExternalWritable := 'False'} : String[4];   // Fourth possible destination
      END_STRUCT;
      si_PLCID { ExternalAccessible := 'False'; ExternalVisible := 'False'; ExternalWritable := 'False'} : Int;   // PLC ID number
      si_FoundPosition { ExternalAccessible := 'False'; ExternalVisible := 'False'; ExternalWritable := 'False'} : Int;   // Character found at this position in string
      si_Gin { ExternalAccessible := 'False'; ExternalVisible := 'False'; ExternalWritable := 'False'} : Int;   // GIN sent by HLC
      sx_HB { ExternalAccessible := 'False'; ExternalVisible := 'False'; ExternalWritable := 'False'} : Bool;   // HB message detect
   END_VAR

   VAR_TEMP
      ti_Position : Int;   // Temporary position parial message
      tx_MsgRead : Bool;   // Message read from FIFO
   END_VAR

   VAR CONSTANT
      cc_DL : Char := '$1D';   // Comma sign
      cs_HB : String := 'HB';   // "HB" message type
      cs_DRespM : String := 'DRespM';   // "DRespM" message type
      cs_GIN : String := 'GIN';   // Gin
   END_VAR


BEGIN
	(*
	----------------------------------------------------------------------------------------

	Version history:
	Date        | Version   | Author        | Remark
	----------------------------------------------------------------------------------------
	18/092/2023 | 4.0       | F.Baten       | First Release TIA 17.5
	*)

	REGION 1 – FIFO header status update

	    // Mode 'S' - FIFO register status update
	    "FC_Fifo"(ic_Mode := 'S',
	              qUDT_Status => #sa_Status.FIFORcvStatus,
	              qx_Error => #sa_Status.FIFOError,
	              qx_Warning => #sa_Status.FIFOWarning,
	              iqv_Data := #sUDT_FifoMsg,
	              iqUDT_FifoHeader := #iqUDT_FifoRcvHeader,
	              iqv_DataBuffer := #iqa_FifoRcvData);

	    IF (NOT #iqUDT_FifoRcvHeader.Status.Empty                               // FIFO not empty
	        AND NOT #sa_Status.FIFOError)                                       // No FIFO error
	    THEN

	        // Mode 'R' - Read FIFO record
	        "FC_Fifo"(ic_Mode := 'R',
	                  qUDT_Status => #sa_Status.FIFORcvStatus,
	                  qx_Error => #sa_Status.FIFOError,
	                  qx_Warning => #sa_Status.FIFOWarning,
	                  iqv_Data := #sUDT_FifoMsg,
	                  iqUDT_FifoHeader := #iqUDT_FifoRcvHeader,
	                  iqv_DataBuffer := #iqa_FifoRcvData);

	        // Message read bit set and position initialize
	        #tx_MsgRead := TRUE;
	        #ti_Position := 0;

	        // FIFO empty or FIFO error occured
	    ELSE

	        #tx_MsgRead := FALSE;

	    END_IF;

	END_REGION


	REGION 2 – Decoding header

	    IF #tx_MsgRead      // New message
	    THEN
	        // Header decode
	        "FC_HMDecodeHeader"(iUDT_FifoMsg := #sUDT_FifoMsg,
	                            qUDT_MSG => #sUDT_MessageHeader);

	        // Check if message was intended for this PLC
	        #si_PLCID := STRING_TO_INT(IN := #sUDT_MessageHeader.PLCID);

	        IF #si_PLCID <> #II_PLCID
	        THEN
	            #tx_MsgRead := FALSE;
	        END_IF;

	    END_IF;

	END_REGION

	REGION 3 - Decoding body

	    IF #tx_MsgRead                                                              // New message
	    THEN
	        // HB
	        IF #sUDT_MessageHeader.MessageHeader = #cs_HB
	        THEN
	            // Faciality ID
	            Chars_TO_Strg(Chars := #sUDT_FifoMsg.Character,
	                          pChars := 31,
	                          Cnt := 9,
	                          Strg => #sa_HBRec."Date");

	            // System ID
	            Chars_TO_Strg(Chars := #sUDT_FifoMsg.Character,
	                          pChars := 40,
	                          Cnt := 12,
	                          Strg => #sa_HBRec."Time");

	            #sx_HB := TRUE;
	        END_IF;

	        IF #sUDT_MessageHeader.MessageHeader = #cs_DRespM
	        THEN

	            // Gin
	            Chars_TO_Strg(Chars := #sUDT_FifoMsg.Character,
	                          pChars := 63,
	                          Cnt := 4,
	                          Strg => #sa_DestRec.Gin);

	            // destination 1
	            Chars_TO_Strg(Chars := #sUDT_FifoMsg.Character,
	                          pChars := 81,
	                          Cnt := 4,
	                          Strg => #sa_DestRec.Dest1);

	            // destination 2
	            Chars_TO_Strg(Chars := #sUDT_FifoMsg.Character,
	                          pChars := 88,
	                          Cnt := 4,
	                          Strg => #sa_DestRec.Dest2);

	            // destination 3
	            Chars_TO_Strg(Chars := #sUDT_FifoMsg.Character,
	                          pChars := 95,
	                          Cnt := 4,
	                          Strg => #sa_DestRec.Dest3);

	            // destination 4
	            Chars_TO_Strg(Chars := #sUDT_FifoMsg.Character,
	                          pChars := 102,
	                          Cnt := 4,
	                          Strg => #sa_DestRec.Dest4);
	        END_IF;

	    END_IF;
	END_REGION

	REGION 4 - Convert and write

	    IF #tx_MsgRead      // New message
	    THEN

	        #si_Gin := STRING_TO_INT(IN := #sa_DestRec.Gin);

	        // Write data from destination assignment message to GIN array
	        IF #si_Gin > 0
	            AND #si_Gin <= 9999
	        THEN
	            IF #sa_DestRec.Dest1 = 'P001' THEN
	                "DB_GIN".GIN[#si_Gin].General.Destination[0] := 1;
	            ELSIF #sa_DestRec.Dest1 = 'P002' THEN
	                "DB_GIN".GIN[#si_Gin].General.Destination[0] := 2;
	            ELSIF #sa_DestRec.Dest1 = 'BOTH' THEN
	                "DB_GIN".GIN[#si_Gin].General.Destination[0] := 3;
	            ELSIF #sa_DestRec.Dest1 = 'NONE' THEN
	                "DB_GIN".GIN[#si_Gin].General.Destination[0] := 99;
	            END_IF;

	            IF #sa_DestRec.Dest2 = 'P001' THEN
	                "DB_GIN".GIN[#si_Gin].General.Destination[1] := 1;
	            ELSIF #sa_DestRec.Dest2 = 'P002' THEN
	                "DB_GIN".GIN[#si_Gin].General.Destination[1] := 2;
	            ELSIF #sa_DestRec.Dest2 = 'BOTH' THEN
	                "DB_GIN".GIN[#si_Gin].General.Destination[1] := 3;
	            ELSIF #sa_DestRec.Dest2 = 'NONE' THEN
	                "DB_GIN".GIN[#si_Gin].General.Destination[1] := 99;
	            END_IF;

	            IF #sa_DestRec.Dest3 = 'P001' THEN
	                "DB_GIN".GIN[#si_Gin].General.Destination[2] := 1;
	            ELSIF #sa_DestRec.Dest3 = 'P002' THEN
	                "DB_GIN".GIN[#si_Gin].General.Destination[2] := 2;
	            ELSIF #sa_DestRec.Dest3 = 'BOTH' THEN
	                "DB_GIN".GIN[#si_Gin].General.Destination[2] := 3;
	            ELSIF #sa_DestRec.Dest3 = 'NONE' THEN
	                "DB_GIN".GIN[#si_Gin].General.Destination[2] := 99;
	            END_IF;

	            IF #sa_DestRec.Dest4 = 'P001' THEN
	                "DB_GIN".GIN[#si_Gin].General.Destination[3] := 1;
	            ELSIF #sa_DestRec.Dest4 = 'P002' THEN
	                "DB_GIN".GIN[#si_Gin].General.Destination[3] := 2;
	            ELSIF #sa_DestRec.Dest4 = 'BOTH' THEN
	                "DB_GIN".GIN[#si_Gin].General.Destination[3] := 3;
	            ELSIF #sa_DestRec.Dest4 = 'NONE' THEN
	                "DB_GIN".GIN[#si_Gin].General.Destination[3] := 99;
	            END_IF;

	        END_IF;

	    END_IF;
	END_REGION













END_FUNCTION_BLOCK

